// TIA Portal V20 export
TYPE "LER_typeAlignSyncMoveMonitoring"
// stored: Access Published
   STRUCT
      error : Bool;
   END_STRUCT;
END_TYPE
